FUNCTION_BLOCK FB_Logger IMPLEMENTS ZigasLibs_Core.I_LoggerEx
VAR
	_fileProperties			: ST_FileProperties;
	_logLevelHeaders		: ZigasLibs_Core.ST_LogLevelHeaders;
	_fileHandler			: FB_FileHandler;
	_events					: ARRAY[0..100] OF Tc2_System.T_MaxString;
	_state					: E_LoggerState;
	_fileExists				: BOOL;
	_localSystemTime		: ZigasLibs_Core.FB_LocalSystemTimeProvider;
	_localSystemTimeString	: Tc2_System.T_MaxString;
	_stringBuilder			: ZigasLibs_Core.FB_StringBuilderBase;
	_bufferFull				: BOOL;
	_amsAddress				: Tc2_System.ST_AmsAddr;
END_VAR

_localSystemTime();
_localSystemTimeString := _localSystemTime.CurrentTimeToString(
	dateSeperator := '.',
	fillWithZeros := TRUE,
	IncludeMilliseconds := FALSE,
	timeFormat := ZigasLibs_Core.E_TimeFormat.YYMMDD_HHMMSS,
	timeOfDaySeperator := ':');

IF _fileHandler.Error THEN
	_state := E_LoggerState.Error;
END_IF

CASE _state OF 
	E_LoggerState.IDLE:
		IF _events[0] <> '' AND _localSystemTime.CurrentTime.IsValid THEN
			_state := E_LoggerState.WRITE_TO_FILE;
		END_IF		
		
	E_LoggerState.WRITE_TO_FILE:
		_fileHandler.FileProperties.FileLocation := _fileProperties.FileLocation;
		_fileHandler.AmsAddress.netId := AmsAddress.netId;
		_fileHandler.FileProperties.FileName := _stringBuilder.Reset()
			.AddString(str := _fileProperties.FileName)
			.AddString(str := TimeForLogName())
			
		
		IF _fileHandler.WriteLine_Append(sContent := _events[0]) AND _fileHandler.Error = FALSE THEN
			THIS^.RemoveEvent();
			_state := E_LoggerState.IDLE;
		END_IF
		
	E_LoggerState.ERROR:
	
END_CASE

METHOD PRIVATE AddLogEntry
VAR_INPUT
	message	: Tc2_System.T_MaxString;
END_VAR

VAR
	i				: ZigasLibs_Core.T_ArrayIndexer;
	eventsMaxIndex	: ZigasLibs_Core.T_ArrayIndexer;
END_VAR
ZigasLibs_Core.ArrayHelper.SetAtFirstEmptySlot(
	arr := _events,
	item := message);

IF _events[100] <> '' THEN
	_bufferFull := TRUE;
ELSE
	_bufferFull := FALSE;
END_IF
END_METHOD

{warning 'add property implementation'}
(* Gets or sets the Ams address structure*)
PROPERTY AmsAddress : REFERENCE TO ZigasLibs_Core.Tc2_System.ST_AmsAddr
GET
AmsAddress ref= _amsAddress;
END_GET
SET
_amsAddress := AmsAddress;
END_SET
END_PROPERTY

PROPERTY PUBLIC BufferFull : BOOL
GET
BufferFull := _bufferFull;
END_GET
END_PROPERTY

(* Gets or set file properties.*)
PROPERTY FileProperties : REFERENCE TO ZigasLibs_Core.ST_FileProperties
GET
FileProperties REF= _fileProperties;
END_GET
SET
_fileProperties := FileProperties;
END_SET
END_PROPERTY

(* Logs the message without any additions.*)
METHOD LogDefault
VAR_INPUT
	message	: ZigasLibs_Core.Tc2_System.T_MaxString;
END_VAR
AddLogEntry(_stringBuilder.Reset() 
	.AddString(str := _localSystemTimeString)
	.AddString(str := ': ')
	.AddString(str := message)
	.Create());
END_METHOD

(* Logs the message by adding the error header to the start.*)
METHOD LogError
VAR_INPUT
	message	: ZigasLibs_Core.Tc2_System.T_MaxString;
END_VAR
AddLogEntry(_stringBuilder.Reset() 
	.AddString(str := _localSystemTimeString)
	.AddString(str := ': ')
	.AddString(str := _logLevelHeaders.Error)
	.AddString(str := message)
	.Create());
END_METHOD

(* Logs the message by adding the info header to the start.*)
METHOD LogInfo
VAR_INPUT
	message	: ZigasLibs_Core.Tc2_System.T_MaxString;
END_VAR
AddLogEntry(_stringBuilder.Reset() 
	.AddString(str := _localSystemTimeString)
	.AddString(str := ': ')
	.AddString(str := _logLevelHeaders.Info)
	.AddString(str := message)
	.Create());
END_METHOD

(* Gets or sets the headers which are applied to logs for their coresponding log levels.*)
PROPERTY LogLevelHeaders : REFERENCE TO ZigasLibs_Core.ST_LogLevelHeaders
GET
LogLevelHeaders ref= _logLevelHeaders;
END_GET
SET
_logLevelHeaders := LogLevelHeaders;
END_SET
END_PROPERTY

(* Logs the message by adding the info header to the start.*)
METHOD LogWarning
VAR_INPUT
	message	: ZigasLibs_Core.Tc2_System.T_MaxString;
END_VAR
AddLogEntry(_stringBuilder.Reset() 
	.AddString(str := _localSystemTimeString)
	.AddString(str := ': ')
	.AddString(str := _logLevelHeaders.Warning)
	.AddString(str := message)
	.Create());
END_METHOD

METHOD RemoveLogEntry
ZigasLibs_Core.ArrayHelper.ShiftDown(
	arr := _events, 
	element := _events[0]);
END_METHOD

METHOD PRIVATE TimeForLogName : STRING
TimeForLogName :=_localSystemTime.CurrentTimeToString(
	timeFormat := ZigasLibs_Core.E_TimeFormat.YYMMDD_HHMMSS,
	timeOfDaySeperator := '_',
	dateSeperator := '',
	fillWithZeros := TRUE,
	IncludeMilliseconds := FALSE)
END_METHOD

END_FUNCTION_BLOCK

(* stored: Version 1.1.0.1, ProductVersion 3.1.4024.13
   POU FB_Logger: Id {86b60fa4-cbc9-0995-00ad-63ce008210aa}, SpecialFunc None
   Folder Private: Id {a06b4692-a5ee-0c61-115f-ec297f5c95cb}
   Folder Methods: Id {860ab4e4-17f1-06ee-0699-9813d104f279}
   Method AddLogEntry: Id {6f1fe8ae-e0ba-067e-058b-4c715ea59a5c}
   Property AmsAddress: Id {2ff23ff9-8aca-06ba-18c7-b3a879ccb01f}
   Get Get: Id {87378494-b48f-041e-0273-a8548009f45b}
   Set Set: Id {03e2518e-8422-04ec-3ebc-7cb2c93733f2}
   Property BufferFull: Id {6b3f66ce-c8e6-0c2b-1325-e4b5c4b64233}
   Get Get: Id {52e4ece1-202f-0628-2423-dc2032edb2da}
   Property FileProperties: Id {673c7f63-7643-01c5-0bc9-18642143b735}
   Get Get: Id {ed145f69-492a-0c2c-1788-7460771a661c}
   Set Set: Id {80c6a351-e367-0411-01ac-b6ae657e0bcb}
   Method LogDefault: Id {03e59e35-6844-0202-3974-90f98220400a}
   Method LogError: Id {60e0135f-a63a-002e-056e-f6dc14cffeb1}
   Method LogInfo: Id {fd97ce6f-9592-08da-013c-a727bade2e2b}
   Property LogLevelHeaders: Id {4a2eeb1a-7fb2-0f80-3c56-845a85555842}
   Get Get: Id {659c25b1-4b2a-01f1-1505-fdb1e25ebd68}
   Set Set: Id {96e644fb-2cc5-081c-3f64-8981e592adf9}
   Method LogWarning: Id {76f0a31c-738d-0885-349f-e0df017a7e19}
   Method RemoveLogEntry: Id {134d7547-21a2-03bc-1ab5-77c94d18ef87}
   Method TimeForLogName: Id {02f4b7c4-160a-013f-0277-3c10823160e9} *)
